FUNCTION_BLOCK HCylinderSA (* Composite Function Block Type *)
  (* Standard: 61499-2 *)
  (* Version 0.0, 9/14/2008, Horst Mayer, nxtControl GmbH, template *)
  PACKAGE Main;
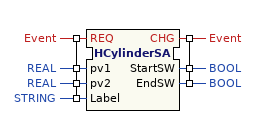
  EVENT_INPUT
    REQ WITH pv1, pv2, Label; (* Normal Execution Request *)
  END_EVENT
  EVENT_OUTPUT
    CHG WITH StartSW, EndSW;
  END_EVENT
  VAR_INPUT
    pv1 : REAL;
    pv2 : REAL;
    Label : STRING;
  END_VAR
  VAR_OUTPUT
    StartSW : BOOL;
    EndSW : BOOL;
  END_VAR
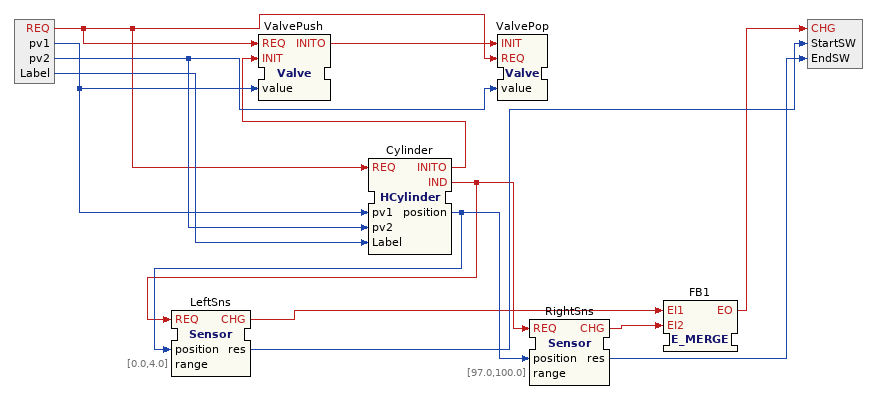
  FBS
    ValvePush : Valve;
    ValvePop : Valve;
    FB1 : E_MERGE;
    LeftSns : Sensor(range := [0.0,4.0]);
    RightSns : Sensor(range := [97.0,100.0]);
    Cylinder : HCylinder;
  END_FBS
  EVENT_CONNECTIONS
    ValvePush.INITO TO ValvePop.INIT;
    FB1.EO TO CHG;
    REQ TO ValvePush.REQ;
    REQ TO ValvePop.REQ;
    LeftSns.CHG TO FB1.EI1;
    RightSns.CHG TO FB1.EI2;
    Cylinder.INITO TO ValvePush.INIT;
    Cylinder.IND TO LeftSns.REQ;
    Cylinder.IND TO RightSns.REQ;
    REQ TO Cylinder.REQ;
  END_CONNECTIONS
  DATA_CONNECTIONS
    pv1 TO ValvePush.value;
    pv2 TO ValvePop.value;
    LeftSns.res TO StartSW;
    RightSns.res TO EndSW;
    Cylinder.position TO LeftSns.position;
    Cylinder.position TO RightSns.position;
    pv1 TO Cylinder.pv1;
    pv2 TO Cylinder.pv2;
    Label TO Cylinder.Label;
  END_CONNECTIONS
END_FUNCTION_BLOCK
